// TIA Portal V16 export
// export: Created 2025-12-18T09:29:18.3028562Z, ExportSetting WithDefaults, DisplayName Totally Integrated Automation Portal, DisplayVersion V16, DisplayName TIA Portal Version Control Interface, DisplayVersion V16, DisplayName TIA Portal Openness, DisplayVersion V16, DisplayName STEP 7 Professional, DisplayVersion V16, DisplayName STEP 7 Safety, DisplayVersion V16, DisplayName WinCC Advanced, DisplayVersion V16
DATA_BLOCK "DB Equipment"   // DB4
{ S7_Optimized_Access := 'TRUE' }
VERSION : 0.1
// stored: AutoNumber true, DBAccessibleFromOPCUA true, IsOnlyStoredInLoadMemory false, IsRetainMemResEnabled false, IsWriteProtectedInAS false, MemoryReserve 100
   VAR
      Station1 : "UDT WorkStation";
      Station2 { S7_SetPoint := 'True'} : "UDT WorkStation";
      Station3 { S7_SetPoint := 'True'} : "UDT WorkStation";
      SupplyStation { S7_SetPoint := 'True'} : "UDT SupplyStation";
   END_VAR
BEGIN
   Station1.Status.tProcessTime := T#0MS;
   Station2.Status.tProcessTime := T#0MS;
   Station3.Status.tProcessTime := T#0MS;
   SupplyStation.Command.xSupplyDataRequest := true;
END_DATA_BLOCK
